// TIA Portal V17 export
// export: Created 2025-03-05T08:02:04.5072038Z, ExportSetting WithDefaults, DisplayName Totally Integrated Automation Portal, DisplayVersion V17 Update 8, DisplayName TIA Portal Openness, DisplayVersion V17 Update 8, DisplayName TIA Portal Version Control Interface, DisplayVersion V17, DisplayName SINAMICS Startdrive Advanced, DisplayVersion V17 SP2, DisplayName SINAMICS Startdrive G110M, G120, G120C, G120D, G120P, G115D, DisplayVersion V17 SP2, DisplayName SINAMICS Startdrive G130, G150, S120, S150, SINAMICS MV, S210, DisplayVersion V17 SP2, DisplayName STEP 7 Professional, DisplayVersion V17 Update 8, DisplayName SINUMERIK ONE STEP 7 Toolbox, DisplayVersion V17 Update 12, DisplayName SINUMERIK 840D sl STEP 7 Toolbox, DisplayVersion V17 Update 12, DisplayName STEP 7 Safety, DisplayVersion V17 Update 6, DisplayName WinCC Advanced, DisplayVersion V17 Update 8
TYPE "LBP_typeModularMcpUniversalOutput"
TITLE = Modular MCP image / Imagen de MCP modulares / Abbild modulare MCP
// Output image of universal keypad for modular MCP / Imagen de salida del panel de mando universal de MCP modulares / Ausgangsabbild des Universal-Bedienfelds für modulare MCP
// stored: IsFailsafeCompliant false
   STRUCT
      led0 : Bool;   // Ausgangsabbild n+0 Bit 0 / output image n+0 bit 0 / Imagen de salida n+0 bit 0
      led1 : Bool;   // Ausgangsabbild n+0 Bit 1 / output image n+0 bit 1 / Imagen de salida n+0 bit 1
      led2 : Bool;   // Ausgangsabbild n+0 Bit 2 / output image n+0 bit 2 / Imagen de salida n+0 bit 2
      led3 : Bool;   // Ausgangsabbild n+0 Bit 3 / output image n+0 bit 3 / Imagen de salida n+0 bit 3
      led4 : Bool;   // Ausgangsabbild n+0 Bit 4 / output image n+0 bit 4 / Imagen de salida n+0 bit 4
      led5 : Bool;   // Ausgangsabbild n+0 Bit 5 / output image n+0 bit 5 / Imagen de salida n+0 bit 5
      led6 : Bool;   // Ausgangsabbild n+0 Bit 6 / output image n+0 bit 6 / Imagen de salida n+0 bit 6
      led7 : Bool;   // Ausgangsabbild n+0 Bit 7 / output image n+0 bit 7 / Imagen de salida n+0 bit 7
      led8 : Bool;   // Ausgangsabbild n+1 Bit 0 / output image n+1 bit 0 / Imagen de salida n+1 bit 0
      led9 : Bool;   // Ausgangsabbild n+1 Bit 1 / output image n+1 bit 1 / Imagen de salida n+1 bit 1
      led10 : Bool;   // Ausgangsabbild n+1 Bit 2 / output image n+1 bit 2 / Imagen de salida n+1 bit 2
      led11 : Bool;   // Ausgangsabbild n+1 Bit 3 / output image n+1 bit 3 / Imagen de salida n+1 bit 3
      led12 : Bool;   // Ausgangsabbild n+1 Bit 4 / output image n+1 bit 4 / Imagen de salida n+1 bit 4
      led13 : Bool;   // Ausgangsabbild n+1 Bit 5 / output image n+1 bit 5 / Imagen de salida n+1 bit 5
      led14 : Bool;   // Ausgangsabbild n+1 Bit 6 / output image n+1 bit 6 / Imagen de salida n+1 bit 6
      reserved17 : Bool;
      led16 : Bool;   // Ausgangsabbild n+2 Bit 0 / output image n+2 bit 0 / Imagen de salida n+2 bit 0
      led17 : Bool;   // Ausgangsabbild n+2 Bit 1 / output image n+2 bit 1 / Imagen de salida n+2 bit 1
      led18 : Bool;   // Ausgangsabbild n+2 Bit 2 / output image n+2 bit 2 / Imagen de salida n+2 bit 2
      reserved23 : Bool;
      reserved24 : Bool;
      reserved25 : Bool;
      reserved26 : Bool;
      reserved27 : Bool;
      led24 : Bool;   // Ausgangsabbild n+3 Bit 0 / output image n+3 bit 0 / Imagen de salida n+3 bit 0
      led25 : Bool;   // Ausgangsabbild n+3 Bit 1 / output image n+3 bit 1 / Imagen de salida n+3 bit 1
      led26 : Bool;   // Ausgangsabbild n+3 Bit 2 / output image n+3 bit 2 / Imagen de salida n+3 bit 2
      reserved33 : Bool;
      reserved34 : Bool;
      reserved35 : Bool;
      reserved36 : Bool;
      reserved37 : Bool;
   END_STRUCT;
END_TYPE
